Fanuc KAREL source: kt00014.KL

-- PROVISIONAL review KL for V770-1; original PC SHA256 5b045d6fc8235037bd6e38f4c0c41edc06bcb85ca19c437c8673c8c237affc94
-- Incomplete behavior may be omitted. Consult companion uncertainty JSON. Do not deploy.
PROGRAM KT00014
%NOLOCKGROUP
VAR
  R1 : REAL
  OUT : REAL
-- UNRESOLVED_DECL Y2 type=002018
BEGIN
  -- UNRESOLVED_PC offsets 5-16; opcodes 2E,23
  -- UNRESOLVED_PC offsets 21-35; opcodes 2E,22,9D,33,B2
  -- UNRESOLVED_PC offsets 40-63; opcodes 21,22,9D,33,B1,64,69,23
  -- UNRESOLVED_PC offsets 68-72; opcodes 7F
END KT00014
